(* CoDeSys 2.3.9.47 project: tank fill and drain.pro *)
(* Libraries: Nexgenie.lib 28.8.18 12:27:24, Standard.lib 28.8.18 12:27:25, Nexgenie_Util.lib 28.8.18 12:27:24, Nexgenie_H.lib 28.8.18 12:27:24, VAW.lib 28.8.18 12:27:25, Modbus.lib 28.8.18 12:27:24 *)

(* PLC configuration (modules and I/O channels)
Nexgenie1000 [Root] node -1, in %IB0 out %QB0
  Nexgenie [Nexgenie] node 0, in %IB0 out %QB0
*)

(* POU PLC_PRG, LD *)
PROGRAM PLC_PRG
VAR
	ON: BOOL;
	STOP: BOOL;
	HL: BOOL;
	X1: BOOL;
	DRAIN: BOOL;
	LL: BOOL;
	X2: BOOL;
	LEVEL: INT;
END_VAR
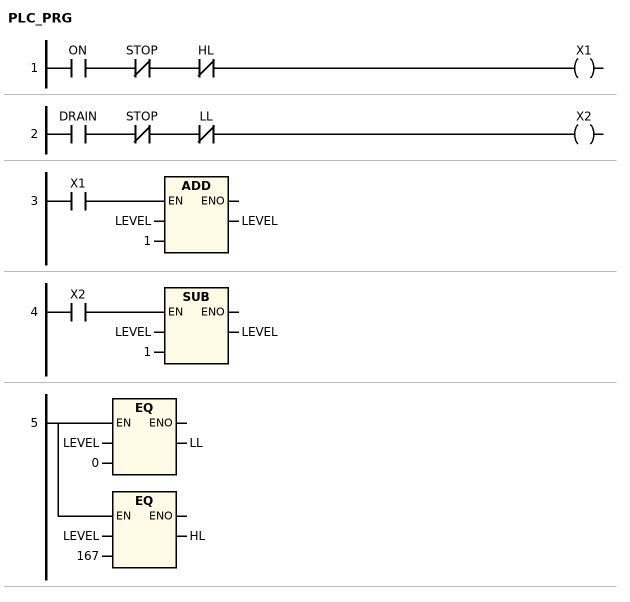
_LD_ (* Ladder Diagram *)
NETWORK 1
	[ON] - [/STOP] - [/HL] --- (X1)
NETWORK 2
	[DRAIN] - [/STOP] - [/LL] --- (X2)
NETWORK 3
	[X1]
		EN --- ADD(LEVEL, 1) => LEVEL
NETWORK 4
	[X2]
		EN --- SUB(LEVEL, 1) => LEVEL
NETWORK 5
	*
		EN --- EQ(LEVEL, 0) => LL
		EN --- EQ(LEVEL, 167) => HL
_END_LD_
(* the same logic as Structured Text *)
(* Network 1 *)
X1 := ON AND NOT STOP AND NOT HL;
(* Network 2 *)
X2 := DRAIN AND NOT (STOP) AND NOT LL;
(* Network 3 *)
IF X1 THEN
	LEVEL := LEVEL + 1;
END_IF;
(* Network 4 *)
IF X2 THEN
	LEVEL := LEVEL - 1;
END_IF;
(* Network 5 *)
LL := LEVEL = 0;
HL := LEVEL = 167;
END_PROGRAM

(* Visualisation LOL
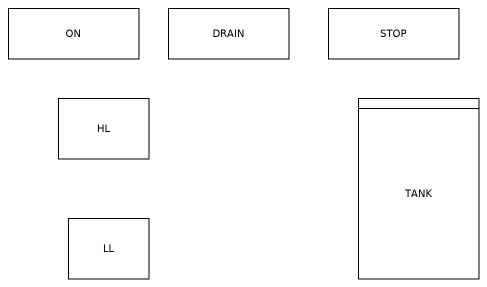
rectangle at (120,40)-(251,91): text "ON"; alarm colour if PLC_PRG.ON; toggles PLC_PRG.ON
rectangle at (280,40)-(401,91): text "DRAIN"; alarm colour if PLC_PRG.DRAIN; toggles PLC_PRG.DRAIN
rectangle at (440,40)-(571,91): text "STOP"; alarm colour if PLC_PRG.STOP; toggles PLC_PRG.STOP
rectangle at (470,140)-(591,311): text "TANK"; alarm colour if PLC_PRG.LEVEL; top 167-PLC_PRG.LEVEL
rounded rectangle at (170,130)-(261,191): text "HL"; alarm colour if PLC_PRG.HL; toggles PLC_PRG.HL
rounded rectangle at (180,250)-(261,311): text "LL"; alarm colour if PLC_PRG.LL; toggles PLC_PRG.LL
1 more shapes without text or variables
*)
